FUNCTION_BLOCK EL2042
VAR
	{attribute addProperty Name "WcState"}
	_wcState : WcStateBase;
	{attribute addProperty Name "Info data"}
	_infoData : InfoDataBase;
	_io : EL2xx2_Data;
END_VAR

PROPERTY IO : REFERENCE TO EL2xx2_Data
GET
IO REF= _io;
END_GET
END_PROPERTY

PROPERTY WcState : REFERENCE TO WcStateBase
GET
WcState REF= _wcState;
END_GET
END_PROPERTY

END_FUNCTION_BLOCK

(* stored: Version 1.1.0.1, ProductVersion 3.1.4024.9
   POU EL2042: Id {04dd3e3c-813a-074c-21ba-2d038e1036a5}, SpecialFunc None
   Property IO: Id {4b45eec2-c31b-09ab-0f88-f35c2ae59824}
   Get Get: Id {de30425c-f824-0449-335d-e7d039e84440}
   Property WcState: Id {fb99a847-1149-07b7-016c-8b319e5860da}
   Get Get: Id {e951e0e2-bb33-0985-32a7-ada990375f48} *)
